FUNCTION_BLOCK TwoConMultiCTL (* Composite Function Block Type *)
  (* Standard: 61499-2 *)
  (* Version 0.2, 2003-12-05, JHC, Rockwell Automation, Renamed from NEWCOMPFB. *)
  (* Version 0.1, 2002-01-08, JHC, Rockwell Automation, Added DLY FB as example. *)
  (* Version 0.0, 2000-05-27, JHC, Rockwell Automation *)
  (* Compiler header: package fb.rt.cs725; *)
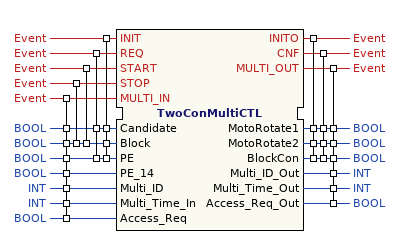
  EVENT_INPUT
    INIT WITH Candidate, Block, PE; (* Initialization Request *)
    REQ WITH Candidate, PE; (* Normal Execution Request *)
    START WITH Block;
    STOP WITH Block;
    MULTI_IN WITH Candidate, Block, PE, PE_14, Multi_ID, Multi_Time_In, Access_Req;
  END_EVENT
  EVENT_OUTPUT
    INITO WITH MotoRotate1, MotoRotate2, BlockCon; (* Initialization Confirm *)
    CNF WITH MotoRotate1, MotoRotate2, BlockCon; (* Execution Confirmation *)
    MULTI_OUT WITH MotoRotate1, MotoRotate2, BlockCon, Multi_ID_Out, Multi_Time_Out, Access_Req_Out;
  END_EVENT
  VAR_INPUT
    Candidate : BOOL;
    Block : BOOL;
    PE : BOOL;
    PE_14 : BOOL;
    Multi_ID : INT;
    Multi_Time_In : INT;
    Access_Req : BOOL;
  END_VAR
  VAR_OUTPUT
    MotoRotate1 : BOOL;
    MotoRotate2 : BOOL;
    BlockCon : BOOL;
    Multi_ID_Out : INT;
    Multi_Time_Out : INT;
    Access_Req_Out : BOOL;
  END_VAR
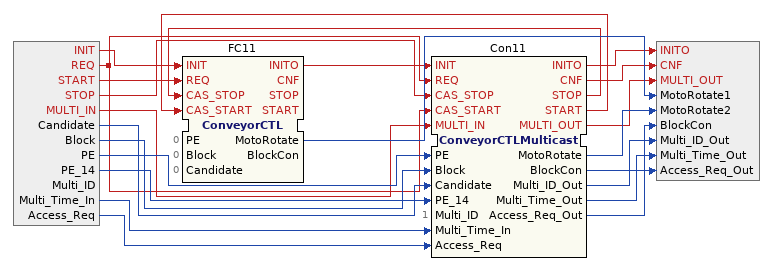
  FBS
    FC11 : ConveyorCTL(PE := 0, Block := 0, Candidate := 0);
    Con11 : ConveyorCTLMulticast(Multi_ID := 1);
  END_FBS
  EVENT_CONNECTIONS
    INIT TO FC11.INIT;
    REQ TO FC11.REQ;
    Con11.INITO TO INITO;
    Con11.CNF TO CNF;
    REQ TO Con11.REQ;
    STOP TO Con11.CAS_STOP;
    START TO Con11.CAS_START;
    Con11.STOP TO FC11.CAS_STOP;
    Con11.START TO FC11.CAS_START;
    FC11.INITO TO Con11.INIT;
    MULTI_IN TO Con11.MULTI_IN;
    Con11.MULTI_OUT TO MULTI_OUT;
  END_CONNECTIONS
  DATA_CONNECTIONS
    Block TO Con11.Block;
    Candidate TO Con11.Candidate;
    PE TO Con11.PE;
    Con11.BlockCon TO BlockCon;
    FC11.MotoRotate TO MotoRotate1;
    Con11.MotoRotate TO MotoRotate2;
    Con11.Multi_ID_Out TO Multi_ID_Out;
    Con11.Multi_Time_Out TO Multi_Time_Out;
    Con11.Access_Req_Out TO Access_Req_Out;
    PE_14 TO Con11.PE_14;
    Multi_Time_In TO Con11.Multi_Time_In;
    Access_Req TO Con11.Access_Req;
  END_CONNECTIONS
END_FUNCTION_BLOCK
